Fanuc TP program (LS listing): MAKRO000.LS

/PROG  MAKRO000
/ATTR
OWNER		= MNEDITOR;
COMMENT		= "A/F_RUECKSETZEN ";
PROG_SIZE	= 2188;
CREATE		= DATE 22-08-03  TIME 07:14:26;
MODIFIED	= DATE 22-08-03  TIME 07:14:26;
FILE_NAME	= ;
VERSION		= 0;
LINE_COUNT	= 111;
MEMORY_SIZE	= 2500;
PROTECT		= READ_WRITE;
STORAGE		= SHADOW;
TCD:  STACK_SIZE	= 0,
      TASK_PRIORITY	= 50,
      TIME_SLICE	= 0,
      BUSY_LAMP_OFF	= 0,
      ABORT_REQUEST	= 0,
      PAUSE_REQUEST	= 0;
DEFAULT_GROUP	= *,*,*,*,*;
CONTROL_CODE	= 00000000 00000000;
/APPL
  SPOT : TRUE ;
  SPOT Welding Equipment Number : 1 ;
/MN
   1:  !Ausgaenge/Flags Ruecksetzen ;
   2:  !KS26 ;
   3:  !Version: 01 ;
   4:  !Stand: 002 ;
   5:  !letzte  Aenderung  06.02.2017 MM ;
   6:  !Warte  bis  PF0 ;
   7:  WAIT (DO[15:OFF])    ;
   8:  !Arbeitsfertigm.  Ruecksetzen ;
   9:  DO[33:OFF]=(OFF) ;
  10:  DO[34:OFF]=(OFF) ;
  11:  DO[35:OFF]=(OFF) ;
  12:  DO[36:OFF]=(OFF) ;
  13:  !Typinfo  Ruecksetzen ;
  14:  DO[37:OFF]=(OFF) ;
  15:  DO[38:OFF]=(OFF) ;
  16:  DO[39:ON ]=(OFF) ;
  17:  DO[40:OFF]=(OFF) ;
  18:  !Roboterverr. Ruecksetzen ;
  19:  DO[41:ON ]=(OFF) ;
  20:  DO[42:ON ]=(OFF) ;
  21:  DO[43:OFF]=(OFF) ;
  22:  DO[44:OFF]=(OFF) ;
  23:  DO[45:ON ]=(OFF) ;
  24:  DO[46:OFF]=(OFF) ;
  25:  DO[47:OFF]=(OFF) ;
  26:  DO[48:OFF]=(OFF) ;
  27:  DO[49:OFF]=(OFF) ;
  28:  DO[50:OFF]=(OFF) ;
  29:  DO[51:OFF]=(OFF) ;
  30:  DO[52:OFF]=(OFF) ;
  31:  DO[53:OFF]=(OFF) ;
  32:  DO[54:OFF]=(OFF) ;
  33:  DO[55:OFF]=(OFF) ;
  34:  DO[56:OFF]=(OFF) ;
  35:  !Werkzeugfreigaben  Ruecksetzen ;
  36:  DO[57:OFF]=(OFF) ;
  37:  DO[58:OFF]=(OFF) ;
  38:  DO[59:OFF]=(OFF) ;
  39:  DO[60:OFF]=(OFF) ;
  40:  DO[61:OFF]=(OFF) ;
  41:  DO[62:ON ]=(OFF) ;
  42:  DO[63:OFF]=(OFF) ;
  43:  DO[64:OFF]=(OFF) ;
  44:  DO[65:OFF]=(OFF) ;
  45:  DO[66:ON ]=(OFF) ;
  46:  DO[67:OFF]=(OFF) ;
  47:  DO[68:OFF]=(OFF) ;
  48:  DO[69:OFF]=(OFF) ;
  49:  DO[70:OFF]=(OFF) ;
  50:  DO[71:ON ]=(OFF) ;
  51:  DO[72:OFF]=(OFF) ;
  52:  DO[73:OFF]=(OFF) ;
  53:  DO[74:OFF]=(OFF) ;
  54:  DO[75:ON ]=(OFF) ;
  55:  DO[76:OFF]=(OFF) ;
  56:  DO[77:ON ]=(OFF) ;
  57:  DO[78:ON ]=(OFF) ;
  58:  DO[79:ON ]=(OFF) ;
  59:  DO[80:ON ]=(OFF) ;
  60:  !Anford. Roboterverr. Ruecksetzen ;
  61:  DO[81:OFF]=(OFF) ;
  62:  DO[82:OFF]=(OFF) ;
  63:  DO[83:OFF]=(OFF) ;
  64:  DO[84:OFF]=(OFF) ;
  65:  DO[85:OFF]=(OFF) ;
  66:  DO[86:OFF]=(OFF) ;
  67:  DO[87:OFF]=(OFF) ;
  68:  DO[88:OFF]=(OFF) ;
  69:  DO[89:OFF]=(OFF) ;
  70:  DO[90:OFF]=(OFF) ;
  71:  DO[91:OFF]=(OFF) ;
  72:  DO[92:OFF]=(OFF) ;
  73:  DO[93:OFF]=(OFF) ;
  74:  DO[94:OFF]=(OFF) ;
  75:  DO[95:OFF]=(OFF) ;
  76:  DO[96:OFF]=(OFF) ;
  77:  !erw. Verriegelungen Ruecksetzen ;
  78:  DO[225:OFF]=(OFF) ;
  79:  DO[226:OFF]=(OFF) ;
  80:  DO[227:OFF]=(OFF) ;
  81:  DO[228:OFF]=(OFF) ;
  82:  DO[229:OFF]=(OFF) ;
  83:  DO[230:OFF]=(OFF) ;
  84:  DO[231:OFF]=(OFF) ;
  85:  DO[232:OFF]=(OFF) ;
  86:  !erw. Typinfo  Ruecksetzen ;
  87:  DO[233:OFF]=(OFF) ;
  88:  DO[234:ON ]=(OFF) ;
  89:  DO[235:OFF]=(OFF) ;
  90:  DO[236:OFF]=(OFF) ;
  91:  DO[237:OFF]=(OFF) ;
  92:  DO[238:OFF]=(OFF) ;
  93:  DO[239:OFF]=(OFF) ;
  94:  DO[240:OFF]=(OFF) ;
  95:  !FRG Ventilsteuerung Ruecksetzen ;
  96:  DO[577:ON ]=(OFF) ;
  97:  DO[701:OFF]=(OFF) ;
  98:  DO[703:OFF]=(OFF) ;
  99:  DO[857:OFF]=(OFF) ;
 100:  DO[2113:OFF]=(OFF) ;
 101:  DO[2121:OFF]=(OFF) ;
 102:  DO[2129:OFF]=(OFF) ;
 103:  DO[2137:OFF]=(OFF) ;
 104:  DO[2145:OFF]=(OFF) ;
 105:  DO[2153:OFF]=(OFF) ;
 106:  DO[2161:OFF]=(OFF) ;
 107:  DO[2169:OFF]=(OFF) ;
 108:  DO[2177:OFF]=(OFF) ;
 109:  DO[2185:OFF]=(OFF) ;
 110:  DO[2193:OFF]=(OFF) ;
 111:  DO[2201:OFF]=(OFF) ;
/POS
/END
